FUNCTION alg_M_mode_a_Dresetled : BOOL
VAR_INPUT
	state: STATE;
END_VAR

alg_M_mode_a_Dresetled := (state.dvar_M_mode) = (elit_reset);

END_FUNCTION

(* stored: Version 1.1.0.1, ProductVersion 3.1.4022.18
   POU alg_M_mode_a_Dresetled: Id {66dcda6a-a5d2-450e-bc29-979a51a349e2}, SpecialFunc None *)
